// SIMATIC S7-200 project (STEP 7-Micro/WIN), CPU 222 CN REL 02.01

ORGANIZATION_BLOCK 主程序:OB1
TITLE=程序注释
// 在一个水泥厂的收尘系统中，这段代码控制“MD-40收尘器”的清灰流程。
// 系统上电时首先进行初始化，复位状态变量并加载参数。操作人员根据收尘器负载的变化，通过清灰间隔选择信号手动设置清灰间隔时间为6000毫秒、12000毫秒或18000毫秒，以适应不同的清灰频率需求。系统通过收尘器运行信号检测收尘器是否在运行，只有当收尘器运行时，系统状态标志才会置位，以支持清灰功能的正常启用。
// 当操作人员通过清灰启动信号触发清灰启动脉冲时，系统进入清灰模式。清灰过程中，清灰周期计数器开始递增至5，以控制脉冲阀1至脉冲阀4的依次动作。脉冲阀1至脉冲阀4在清灰周期计数器的控制下依次开关，每个脉冲阀的喷吹时间由定时器设置为100毫秒，以完成清灰。
// 清灰动作完成后，系统等待清灰间隔时间后再次执行清灰周期。操作人员可以通过清灰停止信号手动结束清灰动作。整个清灰过程依赖系统正常信号的状态，只有在系统正常时才会执行相关操作。
// 
BEGIN
Network 1 // 网络标题
// 网络注释
LD     SM0.4
AN     I0.7
LD     I0.7
O      C0
CTU    C0, +8640
Network 2
LD     C0
LD     I0.7
CTU    C1, +61
Network 3
LD     C1
ON     I0.5
=      M1.0
Network 4
LD     I0.0
=      M0.0
Network 5
LDN    M0.0
ON     I0.5
=      M1.1
Network 6
LD     M1.4
O      M1.6
A      I0.5
=      Q0.0
Network 7
LD     M1.5
O      M1.7
A      I0.5
=      Q0.1
Network 8
LD     M0.0
AN     M1.0
LPS
NOT
JMP    0
LPP
JMP    1
Network 9
LBL    0
Network 10
LD     I0.3
AN     M1.0
EU
=      M1.2
Network 11
LD     M1.2
AN     M1.4
LDN    M1.2
A      M1.4
OLD
A      I0.5
=      M1.4
Network 12
LD     I0.4
AN     M1.0
EU
=      M1.3
Network 13
LD     M1.3
AN     M1.5
LDN    M1.3
A      M1.5
OLD
A      I0.5
=      M1.5
Network 14
LBL    1
Network 15
LD     M0.0
AN     M1.0
=      M3.0
Network 16
LD     M3.0
A      M0.0
A      I0.5
TON    T37, +10
TON    T38, +30
Network 17
LD     M3.0
A      M0.0
LPS
A      T38
=      M1.6
LPP
A      T37
=      M1.7
Network 18
LD     M3.0
A      M0.0
LPS
AN     T40
A      M1.6
TON    T39, +2
LPP
TON    T40, +4
Network 19
LD     M3.0
AN     M0.1
A      M0.3
TON    T41, +10
Network 20
LD     M3.0
A      T41
=      M0.1
Network 21
LD     M3.0
A      M0.0
AN     T46
A      T40
=      M0.2
Network 22
LDN    M0.1
A      M0.2
AN     M0.3
AN     M0.6
TON    T46, +1200
Network 23
LD     M0.2
=      M2.0
TON    T44, +100
A      T44
=      M2.1
TON    T33, +20
Network 24
LD     M0.2
LD     M0.3
O      M1.1
CTU    C2, +5
Network 25
LD     I0.1
AN     I0.2
MOVW   +6000, VW100
Network 26
LDN    I0.1
AN     I0.2
MOVW   +12000, VW100
Network 27
LDN    I0.1
A      I0.2
MOVW   +18000, VW100
Network 28
LD     M0.5
O      M0.6
AN     M0.1
TON    T47, VW100
=      M0.6
Network 29
LDW=   C2, +1
AN     T33
A      M2.1
=      Q0.2
Network 30
LDW=   C2, +2
AN     T33
A      M2.1
=      Q0.3
Network 31
LDW=   C2, +3
AN     T33
A      M2.1
=      Q0.4
Network 32
LDW=   C2, +4
AN     T33
A      M2.1
=      Q0.5
Network 33
LDW=   C2, +5
AN     T33
A      M2.1
=      M0.5
Network 34
LD     M0.3
O      T47
O      T39
AN     M0.1
=      M0.3
END_ORGANIZATION_BLOCK
